FUNCTION_BLOCK FB_PeakshaveBox
VAR_IN_OUT CONSTANT
	st_params 			: ST_peakshavebox_params;
END_VAR

VAR_INPUT
	set					: ST_peakshaveBox_set;
END_VAR

VAR_OUTPUT
	get					: ST_PeakshaveBox_get; 
END_VAR

VAR
	EmptyGet				: ST_PeakshaveBox_get;
	WagoBus					: FB_Wago750354_Buscoupler;
	WagoPQ					: FB_Wago750495_PowerMonitor;
	BeckhoffBus				: FB_EK1100;
	BeckhoffPQ				: FB_EL3453;

	ton_activationDelay		: TON := (PT := T#2S);
END_VAR

VAR_INPUT
	b_enable			: BOOL;
END_VAR

VAR PERSISTENT
	b_BreakerControl 			: BOOL;
	ui_CtRange		 			: UINT := 1000;
	r_VTRatio		 			: REAL := 1;
	b_InverseCTdirection		: BOOL;
END_VAR

ton_activationDelay(IN := get.b_dataOK AND b_enable AND get.b_buscouplerReady, Q => get.b_active);// AND NOT Powermonitor.get.StatusWord.b_Error;
//Instantiate FBs

//PSB settings can only be updated when not active
IF NOT b_enable THEN
	 b_breakerControl := set.b_BreakerControl;
	 ui_ctrange := set.ui_CtRange;
	 r_vtRatio := set.r_VTRatio;
	 b_inverseCTdirection := set.b_InverseCTdirection;
END_IF

get.b_SettingsChangePending := 	(b_breakerControl <> set.b_BreakerControl) OR 
								(ui_ctrange <> set.ui_CtRange) OR 
								(r_vtRatio <> set.r_VTRatio) OR 
								(b_inverseCTdirection <> set.b_InverseCTdirection);
 
CASE st_params.PSBhardware OF
	ePSBHardware.Wago: 
		get.b_dataOK := AcCheck(get.Powermonitor.ar_LineVoltage[0] ,get.Powermonitor.ar_Frequency[0]);
		WagoBus();
		WagoPQ(b_enable:= WagoBus.get.b_SlaveReady, Fastmode := st_params.fastmode, CTinverse := b_InverseCTdirection);
		MapWago();
	ePSBhardware.Beckhoff:
		BeckhoffBus();
		BeckhoffPQ(VoltageRatio := r_VTRatio, CurrentRatio := UINT_TO_INT(ui_CtRange), CTinverse := b_InverseCTdirection);
		MapBeckhoff();	
END_CASE


IF get.b_active THEN
	get.PSBmode := ePSBMode.Monitor;
	IF b_BreakerControl THEN
		get.PSBmode := ePSBMode.MonitorControl;
	END_IF
ELSE
	get.PSBmode := ePSBMode.None;
END_IF

METHOD PUBLIC GetDiagnostics
VAR_IN_OUT
	AddError		: ARRAY [*] OF FB_AddErrorST;
	a_ActiveEvents	: ARRAY [*] OF ST_ErrorStruct;
	w_Index			: WORD;
END_VAR
(*Voltage L1 fault*) 	AddError[w_Index](
			b_ErrorTrig			:= NOT Get.b_buscouplerReady AND b_enable,
			out_ST_Error			:= a_ActiveEvents[w_Index],
			w_ErrorID				:= 1,
			e_ObjectID				:= eObject_ID.PeakshaveBox,
			s_Message				:= 'Buscoupler not detected',
			e_sev					:= eseverity.Warning,
			b_autoClear				:= TRUE
			);
		w_Index := w_Index +1;


(*Voltage L1 fault*) 	AddError[w_Index](
			b_ErrorTrig			:= Get.Powerstatus.b_Error_Phase[1],
			out_ST_Error			:= a_ActiveEvents[w_Index],
			w_ErrorID				:= 2,
			e_ObjectID				:= eObject_ID.PeakshaveBox,
			s_Message				:= 'L1 error',
			e_sev					:= eseverity.Warning,
			b_autoClear				:= TRUE
			);
		w_Index := w_Index +1;
		
(*Voltage L2 fault*) 	AddError[w_Index](
			b_ErrorTrig			:= Get.Powerstatus.b_Error_Phase[2],
			out_ST_Error			:= a_ActiveEvents[w_Index],
			w_ErrorID				:= 3,
			e_ObjectID				:= eObject_ID.PeakshaveBox,
			s_Message				:= 'L2 error',
			e_sev					:= eseverity.Warning,
			b_autoClear				:= TRUE
			);
		w_Index := w_Index +1;
		
(*Voltage L3 fault*) 	AddError[w_Index](
			b_ErrorTrig			:= Get.Powerstatus.b_Error_Phase[3],
			out_ST_Error			:= a_ActiveEvents[w_Index],
			w_ErrorID				:= 4,
			e_ObjectID				:= eObject_ID.PeakshaveBox,
			s_Message				:= 'L3 error',
			e_sev					:= eseverity.Warning,
			b_autoClear				:= TRUE
			);
		w_Index := w_Index +1;
		
(*Powermonitor current L1 out of range*) 	AddError[w_Index](
			b_ErrorTrig			:= Get.PowerStatus.b_OverCurrent AND Get.PowerStatus.b_Error_Phase[1],
			out_ST_Error			:= a_ActiveEvents[w_Index],
			w_ErrorID				:= 6,
			e_ObjectID				:= eObject_ID.PeakshaveBox,
			s_Message				:= 'Powermonitor current L1 out of range',
			e_sev					:= eseverity.Warning,
			b_autoClear				:= TRUE
			);
		w_Index := w_Index +1;
		
(*Powermonitor current L2 out of range*) 	AddError[w_Index](
			b_ErrorTrig			:= Get.PowerStatus.b_OverCurrent AND Get.PowerStatus.b_Error_Phase[2],
			out_ST_Error			:= a_ActiveEvents[w_Index],
			w_ErrorID				:= 7,
			e_ObjectID				:= eObject_ID.PeakshaveBox,
			s_Message				:= 'Powermonitor current L2 out of range',
			e_sev					:= eseverity.Warning,
			b_autoClear				:= TRUE
			);
		w_Index := w_Index +1;
		
(*Powermonitor current L3 out of range*) 	AddError[w_Index](
			b_ErrorTrig			:= Get.PowerStatus.b_OverCurrent AND Get.PowerStatus.b_Error_Phase[3],
			out_ST_Error			:= a_ActiveEvents[w_Index],
			w_ErrorID				:= 8,
			e_ObjectID				:= eObject_ID.PeakshaveBox,
			s_Message				:= 'Powermonitor current L3 out of range',
			e_sev					:= eseverity.Warning,
			b_autoClear				:= TRUE
			);
		w_Index := w_Index +1;
		
(*Powermonitor general warning*) 	AddError[w_Index](
			b_ErrorTrig			:= Get.PowerStatus.b_GeneralWarning,
			out_ST_Error			:= a_ActiveEvents[w_Index],
			w_ErrorID				:= 9,
			e_ObjectID				:= eObject_ID.PeakshaveBox,
			s_Message				:= 'Powermonitor general warning',
			e_sev					:= eseverity.Warning,
			b_autoClear				:= TRUE
			);
		w_Index := w_Index +1;
		

		
(*Powermonitor overcurrent fault*) 	AddError[w_Index](
			b_ErrorTrig				:= Get.PowerStatus.b_OverCurrent,
			out_ST_Error			:= a_ActiveEvents[w_Index],
			w_ErrorID				:= 11,
			e_ObjectID				:= eObject_ID.PeakshaveBox,
			s_Message				:= 'Powermonitor overcurrent fault',
			e_sev					:= eseverity.Warning,
			b_autoClear				:= TRUE
			);
		w_Index := w_Index +1;
		
(*Powermonitor overvoltage fault*) 	AddError[w_Index](
			b_ErrorTrig				:= Get.PowerStatus.b_OverVoltage,
			out_ST_Error			:= a_ActiveEvents[w_Index],
			w_ErrorID				:= 12,
			e_ObjectID				:= eObject_ID.PeakshaveBox,
			s_Message				:= 'Powermonitor overvoltage fault',
			e_sev					:= eseverity.Warning,
			b_autoClear				:= TRUE
			);
		w_Index := w_Index +1;
		
(*Powermonitor undervoltage fault*) 	AddError[w_Index](
			b_ErrorTrig				:= Get.PowerStatus.b_UnderVoltage,
			out_ST_Error			:= a_ActiveEvents[w_Index],
			w_ErrorID				:= 13,
			e_ObjectID				:= eObject_ID.PeakshaveBox,
			s_Message				:= 'Powermonitor undervoltage fault',
			e_sev					:= eseverity.Warning,
			b_autoClear				:= TRUE
			);
		w_Index := w_Index +1;

	
	(*Setting change pending*) 	AddError[w_Index](
			b_ErrorTrig				:= get.b_SettingsChangePending,
			out_ST_Error			:= a_ActiveEvents[w_Index],
			w_ErrorID				:= 14,
			e_ObjectID				:= eObject_ID.PeakshaveBox,
			s_Message				:= 'PSB settings change blocked, disable PSB to apply',
			e_sev					:= eseverity.Warning,
			b_autoClear				:= TRUE
			);
		w_Index := w_Index +1;
END_METHOD

METHOD MapBeckhoff : BOOL

VAR
	i : INT;
END_VAR

VAR_INST
	voltageOK : BOOL;
	currentOK : BOOL;
	PhaseError: BOOL;
END_VAR
get.b_buscouplerReady := beckhoffbus.state = 8 AND beckhoffpq.ui_EL3443BoxState = 8;

IF NOT get.b_buscouplerReady THEN
	get := EmptyGet;	
ELSE
	get.powermonitor.ar_ActivePower := beckhoffPQ.r_ActivePower;
	get.Powermonitor.ar_ApparentPower := beckhoffPQ.r_ApparentPower;
	get.Powermonitor.ar_ReactivePower := beckhoffPQ.r_ReactivePower;
	get.Powermonitor.ar_Current := beckhoffPQ.r_Current;
	get.Powermonitor.ar_LineVoltage := beckhoffPQ.r_LineVoltage;
	get.Powermonitor.ar_PhaseVoltage := beckhoffPQ.r_PhaseVoltage;
	get.powermonitor.ar_Frequency := beckhoffPQ.r_Frequency;
	get.Powermonitor.li_TimeVoltZeroCrossup := beckhoffPQ.li_TimeVoltZeroCrossup;
	//get.Powermonitor.ar_THD := beckhoffPQ
	get.Powermonitor.r_EnergyConsumed := beckhoffPQ.r_ActiveEnergyConsumed;
	get.Powermonitor.r_EnergySupplied:= beckhoffPQ.r_ActiveEnergySupplied;
	get.Powermonitor.r_VoltageUnbalance := beckhoffPQ.r_VoltageUnbalance;
	get.Powermonitor.r_CurrentUnbalance := beckhoffPQ.r_CurrentUnbalance;
	get.Powermonitor.ar_PowerFactor := beckhoffPQ.r_PowerFactor;
	
	get.PowerStatus.b_RotaryField := beckhoffPQ.TotalStatus.bit_GridDirection;
	IF beckhoffPQ.TotalStatus.bit_FrequencyGuardError THEN
		get.Powermonitor.e_ACrotationStatus := eAcrotationstate.None;
	ELSIF beckhoffPQ.TotalStatus.bit_GridDirection THEN
		get.Powermonitor.e_ACrotationStatus := eAcrotationstate.Right;
	ELSE
		get.Powermonitor.e_ACrotationStatus := eAcrotationstate.Left;
	END_IF
	
	
	
	voltageOK := beckhoffPQ.r_LineVoltage[0] <> 0;
	get.PowerStatus.b_OverCurrent := FALSE;
	get.PowerStatus.b_OverVoltage := FALSE;
	get.PowerStatus.b_UnderVoltage := FALSE;
	get.PowerStatus.b_GeneralWarning := 
		beckhoffPQ.TotalStatus.bit_ActivePowerGuardWarning OR
		beckhoffPQ.TotalStatus.bit_ApparentPowerGuardWarning OR
		beckhoffPQ.TotalStatus.bit_FrequencyGuardwarning OR
		beckhoffPQ.TotalStatus.bit_NeutralCurrentGuardWarning OR
		beckhoffPQ.TotalStatus.bit_PowerQualityGuardWarning AND get.b_buscouplerReady;
	get.PowerStatus.b_GeneralFault := 
		beckhoffPQ.TotalStatus.bit_ActivePowerGuardError OR
		beckhoffPQ.TotalStatus.bit_ApparentPowerGuardError OR
		beckhoffPQ.TotalStatus.bit_FrequencyGuardError OR
		beckhoffPQ.TotalStatus.bit_NeutralCurrentGuardError OR
		beckhoffPQ.TotalStatus.bit_PowerQualityGuardError OR
		NOT beckhoffPQ.TotalStatus.bit_SystemState AND get.b_buscouplerReady;
		
	
	//loop through phases 
	FOR i := 1 TO 3 DO
		PhaseError := FALSE;
		CurrentOK := TRUE;
		
		IF beckhoffpq.PhaseStatus[i].bit_VoltageGuardError THEN  
			get.PowerStatus.b_UnderVoltage := TRUE;
			voltageOK := FALSE;	
			PhaseError := TRUE;
		END_IF
		
		IF beckhoffpq.PhaseStatus[i].bit_InaccurateVoltage THEN  
			voltageOK := FALSE;	
			PhaseError := TRUE;
		END_IF
		
		IF beckhoffpq.PhaseStatus[i].bit_Overvoltage THEN
			get.PowerStatus.b_OverVoltage := TRUE;
			voltageOK := FALSE;	
			PhaseError := TRUE;
		END_IF
		
		IF beckhoffpq.PhaseStatus[i].bit_Overcurrent THEN  
			CurrentOK := FALSE;	
			PhaseError := TRUE;
		END_IF
		
		IF beckhoffpq.PhaseStatus[i].bit_Overcurrent THEN
			get.PowerStatus.b_OverCurrent := TRUE;
			CurrentOK := FALSE;
			PhaseError := TRUE;
		END_IF
		
		IF beckhoffPq.PhaseStatus[i].bit_VoltageGuardWarning OR beckhoffPq.PhaseStatus[i].bit_CurrentGuardWarning THEN
			get.PowerStatus.b_GeneralWarning := TRUE;
		END_IF
			
		IF beckhoffPq.PhaseStatus[i].bit_VoltageGuardError OR beckhoffPq.PhaseStatus[i].bit_CurrentGuardError THEN
			get.PowerStatus.b_GeneralFault := TRUE;
			PhaseError := TRUE;
		END_IF
			
		get.PowerStatus.b_Error_Phase[i] := PhaseError;
	END_FOR
	
	get.b_dataOK := VoltageOK AND currentOK AND beckhoffPQ.TotalStatus.bit_SystemState;
END_IF
END_METHOD

METHOD MapWago : BOOL
VAR_INPUT
END_VAR
get.b_buscouplerReady := wagobus.get.b_SlaveReady;

IF NOT get.b_buscouplerReady THEN
	get := EmptyGet;	
ELSE
	get.Powermonitor.ar_ActivePower := WagoPQ.get.Data.ar_ActivePower;
	get.Powermonitor.ar_ReactivePower := WagoPQ.get.Data.ar_ReactivePower;
	get.Powermonitor.ar_ApparentPower := WagoPQ.get.Data.ar_ApparentPower;
	get.Powermonitor.ar_Current := WagoPQ.get.Data.ar_CurrentRMS;
	get.Powermonitor.ar_LineVoltage := WagoPQ.get.Data.ar_VoltageLL;
	get.Powermonitor.ar_PhaseVoltage := WagoPQ.get.Data.ar_VoltageLN;
	get.powermonitor.ar_Frequency := WagoPQ.get.Data.ar_Frequency;
	//get.Powermonitor.ar_THD := beckhoffPQ
	get.Powermonitor.r_EnergyConsumed := WagoPQ.get.Data.r_ActiveEnergyImport;
	get.Powermonitor.r_EnergySupplied:= WagoPQ.get.Data.r_ActiveEnergyExport;
	get.Powermonitor.r_VoltageUnbalance := 0;
	get.Powermonitor.r_CurrentUnbalance := 0;
	get.Powermonitor.ar_PowerFactor := wagoPQ.get.Data.ar_Powerfactor;
	
	get.PowerStatus.b_Error_Phase[1] := wagoPQ.get.StatusWord.b_Error_L1;
	get.PowerStatus.b_Error_Phase[2] := wagoPQ.get.StatusWord.b_Error_L2;
	get.PowerStatus.b_Error_Phase[3] := wagoPQ.get.StatusWord.b_Error_L3;
	get.PowerStatus.b_OverCurrent := wagoPQ.get.ExtStatusWord.b_OverCurrent;
	get.PowerStatus.b_OverVoltage := wagoPQ.get.ExtStatusWord.b_OverVoltage;
	get.PowerStatus.b_RotaryField := wagoPQ.get.ExtStatusWord.b_RotaryField;
	get.PowerStatus.b_GeneralFault := wagoPQ.get.StatusWord.b_Error;
	get.PowerStatus.b_GeneralWarning := wagoPQ.get.StatusWord.b_Warning;
	
	IF get.PowerStatus.b_GeneralFault THEN
		get.Powermonitor.e_ACrotationStatus := eAcrotationstate.None;
	ELSIF beckhoffPQ.TotalStatus.bit_GridDirection THEN
		get.Powermonitor.e_ACrotationStatus := eAcrotationstate.Right;
	ELSE
		get.Powermonitor.e_ACrotationStatus := eAcrotationstate.Left;
	END_IF
END_IF
END_METHOD

END_FUNCTION_BLOCK

(* stored: Version 1.1.0.1, ProductVersion 3.1.4024.12
   POU FB_PeakshaveBox: Id {be0f6613-070e-4d0b-a99d-ae5163fe483c}, SpecialFunc None
   Method GetDiagnostics: Id {d4bb2571-9c0f-41d6-947c-974663bd2041}
   Method MapBeckhoff: Id {3fe9e893-a947-4ebc-a260-f374e67c0f13}
   Method MapWago: Id {6d533cf0-8412-46fa-ae9e-213721a90df6} *)
